FUNCTION_BLOCK "FB_DI"
TITLE = Func Block from DI
{ S7_Optimized_Access := 'FALSE' }
VERSION : 1.2
// ==============================================================================
// Файл: S7C_FC_Filter_PT1.scl
// Целевые ПЛК: S7-1200 / S7-1500 (Линейка Current)
// Особенности:
// - Оптимизированный доступ (Optimized block access = TRUE)
// - Использование современных системных функций (время цикла, первый скан)
// - Кодировка при сохранении: UTF-8 with BOM
// ==============================================================================
   VAR_INPUT
      i_boRaw { ExternalAccessible := 'False'; ExternalVisible := 'False'; ExternalWritable := 'False'} : Bool;   // Сырой физический вход
   END_VAR

   VAR_IN_OUT
      io_stConfig : "UDT_DI_Conf";
      io_stOut : "UDT_DI_Out";
   END_VAR

   VAR
      stat_TonFlt {InstructionName := 'TON_TIME'; LibVersion := '1.0'; ExternalAccessible := 'False'; ExternalVisible := 'False'; ExternalWritable := 'False'; S7_SetPoint := 'False'} : TON_TIME;   // Задержка включения
      stat_TofFlt {InstructionName := 'TOF_TIME'; LibVersion := '1.0'; ExternalAccessible := 'False'; ExternalVisible := 'False'; ExternalWritable := 'False'; S7_SetPoint := 'False'} : TOF_TIME;   // Задержка выключения
      stat_Mode { ExternalAccessible := 'False'; ExternalVisible := 'False'; ExternalWritable := 'False'} : Int;   // Текущий рабочий режим
      stat_OldMode { ExternalAccessible := 'False'; ExternalVisible := 'False'; ExternalWritable := 'False'} : Int;   // Предыдущий режим для отслеживания изменений
   END_VAR

   VAR_TEMP
      temp_FilterTime : Time;
      temp_boDisabled : Bool;
      temp_boNorm : Bool;
      temp_boInvert : Bool;
   END_VAR


BEGIN

	    #temp_boDisabled := (#io_stConfig.Mode = "DB_Global".c_stDI_Mode.Disabled);

	    IF #temp_boDisabled THEN
	        #stat_Mode := "DB_Global".c_stDI_Mode.None;
	        RETURN;
	    END_IF;

	    // =========================================================
	    // 1. ПРОВЕРКА РЕЖИМА И ПРЕОБРАЗОВАНИЕ ВРЕМЕНИ
	    // =========================================================
	    #stat_Mode := #io_stConfig.Mode;

	    IF #stat_Mode < 0 OR #stat_Mode > "DB_Global".c_stDI_Mode.Disabled THEN
	        #stat_Mode := "DB_Global".c_stDI_Mode.None;
	    END_IF;

	    // Преобразуем мс (Int) в формат Time
	    #temp_FilterTime := DINT_TO_TIME(INT_TO_DINT(#io_stConfig.FilterTime));

	    // =========================================================
	    // 2. СБРОС ТАЙМЕРОВ ПРИ СМЕНЕ РЕЖИМА
	    // =========================================================
	    IF #stat_Mode <> #stat_OldMode THEN
	        #stat_TonFlt(IN := FALSE,
	                     PT := #temp_FilterTime);
	        #stat_TofFlt(IN := FALSE,
	                     PT := #temp_FilterTime);

	        #io_stOut.Value := #i_boRaw;
	        #stat_OldMode := #stat_Mode;
	    END_IF;

	    // =========================================================
	    // 3. ЛОГИКА ФИЛЬТРАЦИИ И ИНВЕРСИИ
	    // =========================================================
	    IF #stat_Mode = "DB_Global".c_stDI_Mode.None THEN
	        // Режим 0: Прямая передача сигнала (без фильтра)
	        #io_stOut.Value := #i_boRaw;

	        // Сбрасываем таймеры, чтобы они не висели в фоне
	        #stat_TonFlt(IN := FALSE,
	                     PT := #temp_FilterTime);
	        #stat_TofFlt(IN := FALSE,
	                     PT := #temp_FilterTime);

	    ELSE
	        // Режимы с фильтром: применяем TON и TOF
	        #stat_TonFlt(IN := #i_boRaw,
	                     PT := #temp_FilterTime);
	        #stat_TofFlt(IN := #i_boRaw,
	                     PT := #temp_FilterTime);

	        // Включение (TON отработал) -> сигнал стабильно TRUE
	        IF #stat_TonFlt.Q THEN
	            #io_stOut.Value := (#stat_Mode = "DB_Global".c_stDI_Mode.NOpen);
	        END_IF;

	        // Выключение (TOF отработал) -> сигнал стабильно FALSE
	        IF NOT #stat_TofFlt.Q THEN
	            #io_stOut.Value := (#stat_Mode <> "DB_Global".c_stDI_Mode.NOpen); // Сбрасываем соответственно режиму
	        END_IF;
	    END_IF;

END_FUNCTION_BLOCK

